FUNCTION_BLOCK MemoOC (* Basic Function Block Type *)
  (* Standard: 61499-2 *)
  (* Version 0.0, 8/17/2026, Schneider Electric, Template *)
  PACKAGE SE.Nereda;
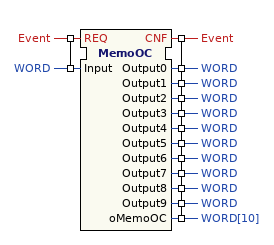
  EVENT_INPUT
    REQ WITH Input; (* Normal Execution Request *)
  END_EVENT
  EVENT_OUTPUT
    CNF WITH Output0, Output1, Output2, Output3, Output4, Output5, Output6, Output7, Output8, Output9, oMemoOC; (* Execution Confirmation *)
  END_EVENT
  VAR_INPUT
    Input : WORD;
  END_VAR
  VAR_OUTPUT
    Output0 : WORD;
    Output1 : WORD;
    Output2 : WORD;
    Output3 : WORD;
    Output4 : WORD;
    Output5 : WORD;
    Output6 : WORD;
    Output7 : WORD;
    Output8 : WORD;
    Output9 : WORD;
    oMemoOC : ARRAY [0..9] OF WORD;
  END_VAR
  VAR
    MemoOC : ARRAY [0..9] OF WORD;
    i : INT := 0;
  END_VAR
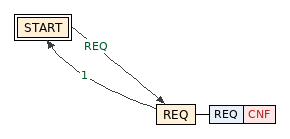
  EC_STATES
    START; (* Initial State *)
    REQ : REQ -> CNF; (* Normal execution *)
  END_STATES
  EC_TRANSITIONS
    START TO REQ := REQ;
    REQ TO START := 1;
  END_TRANSITIONS
  ALGORITHM REQ IN ST: (* Normally executed algorithm *)
;
FOR i := 8 TO 0 BY -1 DO
    MemoOC[i + 1] := MemoOC[i];
END_FOR;

MemoOC[0] := Input;

Output0 := MemoOC[0];
Output1 := MemoOC[1];
Output2 := MemoOC[2];
Output3 := MemoOC[3];
Output4 := MemoOC[4];
Output5 := MemoOC[5];
Output6 := MemoOC[6];
Output7 := MemoOC[7];
Output8 := MemoOC[8];
Output9 := MemoOC[9];

oMemoOC := MemoOC;
  END_ALGORITHM
END_FUNCTION_BLOCK
